// TIA Portal V17 export
// export: Created 2024-09-02T12:50:30.6927006Z, ExportSetting WithDefaults, DisplayName Totally Integrated Automation Portal, DisplayVersion V17, DisplayName TIA Portal Openness, DisplayVersion V17, DisplayName TIA Portal Version Control Interface, DisplayVersion V17, DisplayName STEP 7 Professional, DisplayVersion V17, DisplayName STEP 7 Safety, DisplayVersion V17, DisplayName WinCC Professional, DisplayVersion V17
TYPE "type_Cognex_DM"
// stored: IsFailsafeCompliant false
   STRUCT
      HMI : Struct   // HMI-Button
         FrgFkt : Struct   // Freigabe / Approve
            Gestaltung : Int;   // Button Anzeige Gestaltung / Button Display Design
            aktiv : Bool;   // Button aktiv (gedrückt) / Button active (pressed)
         END_STRUCT;
         Reset : Struct   // Button "Reset"
            Gestaltung : Int;   // Button Anzeige Gestaltung / Button Display Design
            aktiv : Bool;   // Button aktiv (gedrückt) / Button active (pressed)
         END_STRUCT;
         Read : Struct   // Button "Read"
            Gestaltung : Int;   // Button Anzeige Gestaltung / Button Display Design
            aktiv : Bool;   // Button aktiv (gedrückt) / Button active (pressed)
         END_STRUCT;
         SetPrg : Struct   // Button "Set Programm"
            Gestaltung : Int;   // Button Anzeige Gestaltung / Button Display Design
            aktiv : Bool;   // Button aktiv (gedrückt) / Button active (pressed)
         END_STRUCT;
         Write : Struct   // Button "Write"
            Gestaltung : Int;   // Button Anzeige Gestaltung / Button Display Design
            aktiv : Bool;   // Button aktiv (gedrückt) / Button active (pressed)
         END_STRUCT;
         Lighting : Struct   // Button "Lighting"
            Gestaltung : Int;   // Button Anzeige Gestaltung / Button Display Design
            aktiv : Bool;   // Button aktiv (gedrückt) / Button active (pressed)
         END_STRUCT;
         ResetStatistik : Struct   // Button "Statistik Reset"
            Gestaltung : Int;   // Button Anzeige Gestaltung / Button Display Design
            aktiv : Bool;   // Button aktiv (gedrückt) / Button active (pressed)
         END_STRUCT;
         Res_07 : Struct   // Button " "
            Gestaltung : Int;   // Button Anzeige Gestaltung / Button Display Design
            aktiv : Bool;   // Button aktiv (gedrückt) / Button active (pressed)
         END_STRUCT;
         Res_08 : Struct   // Button " "
            Gestaltung : Int;   // Button Anzeige Gestaltung / Button Display Design
            aktiv : Bool;   // Button aktiv (gedrückt) / Button active (pressed)
         END_STRUCT;
         ProgNbr { S7_SetPoint := 'True'} : Int := 1;   // Program number for reset operation (default "1")
      END_STRUCT;
      Anzeige { ExternalWritable := 'False'} : Struct   // Anzeige / Display
         StatusBool { ExternalWritable := 'False'} : DWord;   // Status
         StatusInt { ExternalWritable := 'False'} : Array[0..5] of Int;   // Status ID / status ID
         Ergebnis { ExternalWritable := 'False'} : Array[0..7] of LInt;   // Statistik / Statistics
      END_STRUCT;
      Start { ExternalWritable := 'False'} : Bool;   // Start
      Reset { ExternalWritable := 'False'} : Bool;   // Reset
      Licht { ExternalWritable := 'False'} : Bool;   // Licht ein / Light on
      DoneOk { ExternalWritable := 'False'} : Bool;   // DM Fertig IO / DM Ready OK
      DoneNOk { ExternalWritable := 'False'} : Bool;   // DM Fertig NIO / DM Ready NOK
      Done { ExternalWritable := 'False'} : Bool;   // Hand Scanner Done
      Error { ExternalWritable := 'False'} : Byte;   // Result error in written result (match error, read error) / Result error in written result (match error, read error)
      ProgNr { ExternalWritable := 'False'} : Int;   // Programmnummer / program number
      ResultQ { ExternalWritable := 'False'} : Char;   // Code quality / Code quality
      ResultLn { ExternalWritable := 'False'} : Int;   // Anzahl Daten / Number of data:
      ResultStr { ExternalWritable := 'False'} : String;   // Daten in String / Data in string
      ResultChar { ExternalWritable := 'False'} : Array[1..246] of Char;   // Daten in Char / Data in Char
   END_STRUCT;
END_TYPE
